{attribute addProperty BoxType "ER1258-0001-0019"}
{attribute addProperty Id "ChannelAT %I*ARRAY[0..7] OF Channel_E4AEF59E6480LatchAT %I*Latch_54D9ECC2272340WcStateAT %I*WcState_C1B70B0F3240InfoDataAT %I*InfoData_7231B2DD80100"}
{attribute addProperty CRC "3111238133"}
{attribute addProperty SizeInBites "448"}
{attribute addProperty SizeInBytes "56"}
TYPE ER1258_402FC40E :
STRUCT
	{attribute addProperty Name "Channel"}
	Channel : ARRAY[0..7] OF Channel_E4AEF59E;
	{attribute addProperty Name "Latch"}
	Latch : Latch_54D9ECC2;
	{attribute addProperty Name "WcState"}
	WcState : WcState_C1B70B0F;
	{attribute addProperty Name "InfoData"}
	InfoData : InfoData_7231B2DD;
END_STRUCT
END_TYPE

(* stored: Version 1.2.0.0, ProductVersion 3.1.4024.9
   DUT ER1258_402FC40E: Id {0aa34757-205a-4052-ab62-c6833f6e8418} *)
